FUNCTION_BLOCK FB_SimpleTest IMPLEMENTS ITest
VAR_INPUT
END_VAR
VAR_OUTPUT
END_VAR
VAR
	stResult		: TestResults;
	sName			: STRING;
	sClassName		: STRING := __POUNAME();
END_VAR

METHOD PROTECTED AssertEquals
VAR_INPUT
	expected		: ANY;
	result			: ANY;
	failmsg			: STRING(255);
END_VAR
VAR
	sExp, sRes		: STRING;
END_VAR
IF (expected.diSize <> result.diSize) THEN
	stResult.Message := 'Test error: expected value type mismatch';
	stResult.Passed := FALSE;
	RETURN;
END_IF

IF (Expected.pValue^ <> Result.pValue^) THEN
	sExp := CONCAT(' Expected: ', TO_STRING(expected.pValue^));
	sRes := CONCAT(' Result: ', TO_STRING(result.pValue^));
	stResult.Message := CONCAT(CONCAT(failmsg, sExp), sRes);
	stResult.Passed := FALSE;
ELSE
	stResult.Passed := TRUE;
END_IF
END_METHOD

PROPERTY ClassName : STRING
GET
ClassName := sClassName;
END_GET
END_PROPERTY

METHOD Execute : BOOL
VAR_INPUT
END_VAR
END_METHOD

//FB_Init is always available implicitly and it is used primarily for initialization.
//The return value is not evaluated. For a specific influence, you can also declare the
//methods explicitly and provide additional code there with the standard initialization
//code. You can evaluate the return value.
METHOD FB_Init: BOOL
VAR_INPUT
    bInitRetains: BOOL; // TRUE: the retain variables are initialized (reset warm / reset cold)
    bInCopyCode: BOOL;  // TRUE: the instance will be copied to the copy code afterward (online change) 
	sTestName : STRING;
END_VAR
THIS^.sName := sName;
END_METHOD

PROPERTY Name : STRING
GET
Name := sName;
END_GET
END_PROPERTY

PROPERTY Result : TestResults
GET
Result := stResult;
END_GET
END_PROPERTY

END_FUNCTION_BLOCK

(* stored: Version 1.1.0.1
   POU FB_SimpleTest: Id {a76d9921-ad37-4ebf-aed3-d89b8cd7a1ee}, SpecialFunc None
   Method AssertEquals: Id {585f4c2a-8ee9-4688-8bda-614a35dedf4a}
   Property ClassName: Id {911d440e-ce97-493d-abf6-a059f8ab03fd}
   Get Get: Id {faf3cdf4-1d51-4306-a52a-f97533db893a}
   Method Execute: Id {d3694038-a5af-4a33-9a56-6eccc4378ffd}
   Method FB_init: Id {51e04b6e-3325-40a5-a8fb-82f6ed372341}
   Property Name: Id {2be2eac5-7a6f-4456-b3b3-8cb86688f8a4}
   Get Get: Id {68516f1e-cfb6-4e16-9df6-dead141c721b}
   Property Result: Id {3b92dccb-6945-4c38-8cd7-a1313895bf93}
   Get Get: Id {64227010-83a2-4c08-b100-a928a84aa30f} *)
